FUNCTION_BLOCK ControlValv_ioLink
VAR_INPUT
	Comando:BOOL;
	Status_1:BYTE;
	Teste:BOOL:=FALSE;
	Inverter:BOOL;
	PosicaoIN:INT;		//Posição da válvula. Valor vindo do IOLink
END_VAR
VAR_OUTPUT
	Estado:INT;
	Falla:BOOL;
	END_VAR
VAR_IN_OUT
	Actuar:BYTE;
END_VAR
VAR
	TemposAcionamento	:ARRAY[1..10] OF DINT;	//Array com os últimos tempos de acionamento
	SwitchCase: INT;
	RTrig: R_TRIG;
	TON_Acionamento: TON;
	iCounter: INT;
	TON_Teste: TON;
	ResetContagem: BOOL;
	PosicaoOUT	:REAL;	//Posição da válvula convertida em %
	IniciarCfg	:BOOL;	//Se a válvula estiver aberta e esse comando for dado, salva o valor de posição como 100%. O mesmo para ela fechada
END_VAR

VAR PERSISTENT
	qntAcionamentos:DINT;	//Quantidade de acionamentos da válvula
	cfgPosicao	:DUT_cfgPosicValvula;		//Configuração de conversão do posicionamento das válvulas
	UltimasPosicoes	:ARRAY[1..2] OF REAL;	//Esse array salva as últimas posições de abertura e fechamento [1] - Abertura, [2] - Fechamento
	
END_VAR

//Acionamento da válvula
Actuar.04 := (Comando AND NOT Inverter) OR (NOT Comando AND Inverter) OR (Teste AND AquecimentoValvulas.Acionar);

TON_Teste(IN:= Actuar.04, PT:= T#465MS);

//Se não estiver em teste, verifica se está aberta, fechada ou em falha
IF NOT Teste THEN
	IF Status_1.0 = 1 THEN	//Válvula aberta
		Estado := 2;
		UltimasPosicoes[1] := PosicaoOUT;	//Salva a posição da válvula no array
	END_IF
	IF Status_1.1 = 1 THEN	//Válvula fechada
		Estado := 1;
		UltimasPosicoes[2] := PosicaoOUT;	//Salva a posição da válvula no array
	END_IF
	IF Status_1.4 = 1 THEN	//Em falha
		Falla := 1;
		Estado := 6;
	END_IF
ELSE
	IF TON_Teste.Q THEN
		Estado := 1;
	ELSE
		Estado := 2;
	END_IF
END_IF

//A lógica abaixo foi feita para calcular o tempo de acionamento da válvula
//Detecta a borda de subida do comando de acionamento
RTrig(CLK:= Actuar.04, Q=> );


//Temporizador do acionamento
TON_Acionamento(IN:= , PT:= T#1M, Q=> , ET=> );

//Se a borda for detectada, inicia a máquina de estados
IF RTRIG.Q THEN
	SwitchCase := 1;
	TON_Acionamento.IN := TRUE;
	//Incrementa os acionamentos
	qntAcionamentos := qntAcionamentos + 1;
END_IF

//Reset da contagem de acionamentos
IF ResetContagem THEN
	qntAcionamentos := 0;
	ResetContagem := FALSE;
END_IF

//Temporizador do acionamento
TON_Acionamento(IN:= , PT:= , Q=> , ET=> );

//Cancela o cálculo se a válvula entrar em falha
IF Falla THEN
	SwitchCase := 0;
END_IF

CASE SwitchCase OF
	1:	IF Estado = 2 THEN
			TemposAcionamento[10] := TIME_TO_DINT(TON_Acionamento.ET);
			SwitchCase := 2;
		END_IF
		
	2:	FOR iCounter := 1 TO 9 BY 1 DO 
			TemposAcionamento[iCounter] := TemposAcionamento[iCounter + 1];
		END_FOR
		TON_Acionamento.IN := FALSE;
		SwitchCase := 0;
END_CASE

//Se a válvula estiver aberta e esse comando for dado, salva o valor de posição como 100%. O mesmo para ela fechada
IF IniciarCfg THEN
	IF Estado = 2 THEN
		cfgPosicao.Aberta := PosicaoIN;
	ELSIF Estado = 1 THEN
		cfgPosicao.Fechada := PosicaoIN;
	END_IF;
	IniciarCfg := FALSE;
END_IF

PosicaoOUT := SEL((cfgPosicao.Aberta - cfgPosicao.Fechada) <> 0,0,(100/(TO_REAL(cfgPosicao.Aberta - cfgPosicao.Fechada))) * (PosicaoIN - cfgPosicao.Fechada));

END_FUNCTION_BLOCK

(* stored: Version 1.1.0.1, ProductVersion 3.1.4024.14
   POU ControlValv_ioLink: Id {2557b125-896a-4d9a-b8fa-f53da0f1731a}, SpecialFunc None *)
